Universal Robots PolyScope program: Subprogram .urp

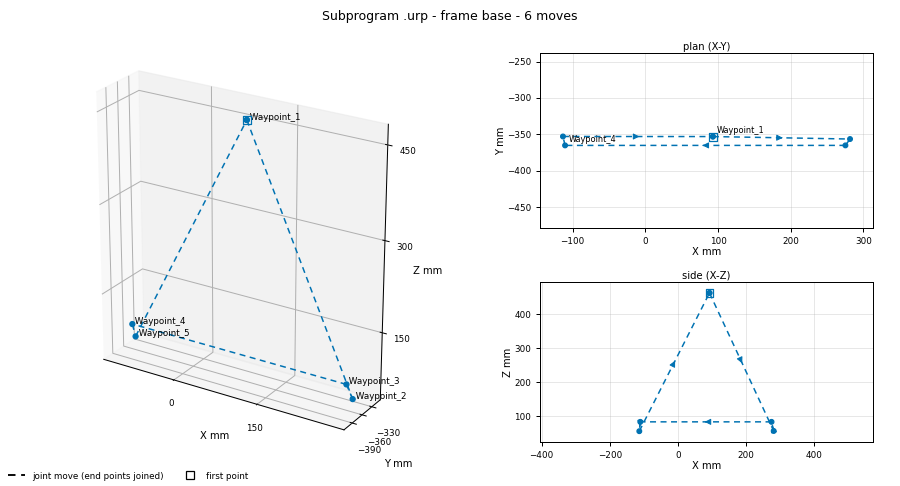
[picture p0: tool path of Subprogram .urp in frame base, 6 of 6 moves have a stored position in this frame; points joined in program order, loops and branches not executed]
Program PythonSubprogram  (installation=default directory=/programs/usbdisk/NoodleBotSoftware createdIn=3.12.1.90940 lastSavedIn=3.12.1.90940 robotSerialNumber=2017354841)
Calibrated DH parameters: a=[0.000094, -0.006117, -0.382762, 0.000086, 0.000044, 0]; d=[0.089236, 217.751846, -204.357806, -13.283746, 0.094902, 0.082641]; alpha=[1.57017, 0.001953, -0.006493, 1.570192, -1.570543, 0]; deltaTheta=[0.000036, 1.556386, -1.779789, 0.223359, -0.000014, -0.000001]
BeforeStart
  var_1 := socket_open("192.168.0.100",30000)
Robot Program (runOnlyOnce=false)
  Loop While (checkContinuously=false) expression=var_1≟ False
    var_1 := socket_open("192.168.0.100",30000)
    Wait Sleep waitTime=0.5
  Script: socket_send_string("asking_for_data")
  Wait Sleep waitTime=0.5
  var_2 := socket_read_ascii_float(1)
  Wait Sleep waitTime=0.5
  var_1 := False
  Script: socket_close()
  If var_2[0]≟1
    Call Test_ur5a
SubProgram -> Test_ur5a
SubProgram Test_ur5a (keepSynchronizedWithDisk=false) programFile=/programs/Test ur5a.urp
  MoveJ speed 60 deg/s, acceleration 80 deg/s^2 (useActiveTCP=true)
    URCap RG2 (RG - On Robot, OnRobot A/S) dataModel(depthCompensate=false, force=40, payload=0.0, width=86, name=RG2(86))
    Waypoint Waypoint_1: TCP in base x=92.939 y=-353.097 z=462.595 mm, rx=1.1692 ry=-1.2408 rz=1.1709 rad; joints [88.542, -137.018, 138.65, 178.588, 268.341, 89.999] deg; flange x=103.097 y=-166.778 z=463.297 mm, rx=1.2543 ry=1.1818 rz=-1.2438 rad
    Wait Sleep waitTime=1
    Waypoint Waypoint_2: TCP in base x=281.568 y=-356.493 z=57.062 mm, rx=2.4509 ry=-1.0812 rz=-0.3973 rad; joints [131.142, -83.255, 116.241, 241.937, 240.139, 90.003] deg; flange x=360.116 y=-306.414 z=218.729 mm, rx=-1.1245 ry=-2.5488 rz=0.6202 rad
    URCap RG2 (RG - On Robot, OnRobot A/S) dataModel(depthCompensate=false, payload=0.0, force=40, width=0, name=RG2(0))
    Wait Sleep waitTime=1
    Waypoint Waypoint_3: motionParameters(jointSpeed=1.745329 jointAcceleration=4.363323 cartesianSpeed=0.25 cartesianAcceleration=1.2); TCP in base x=275.23 y=-365.244 z=83.858 mm, rx=2.4082 ry=-1.0628 rz=-0.4074 rad; joints [131.131, -84.8, 114.576, 244.685, 237.533, 90.016] deg; flange x=358.189 y=-309.185 z=241.34 mm, rx=-1.1149 ry=-2.5256 rz=0.6807 rad
    Wait Sleep waitTime=1
    Waypoint Waypoint_4: motionParameters(jointSpeed=1.745329 jointAcceleration=4.363323 cartesianSpeed=0.25 cartesianAcceleration=1.2); TCP in base x=-110.35 y=-365.263 z=83.889 mm, rx=2.4083 ry=-1.0627 rz=-0.4074 rad; joints [69.173, -109.993, 144.496, 207.947, 251.859, 22.112] deg; flange x=-27.414 y=-309.154 z=241.302 mm, rx=-1.1146 ry=-2.5256 rz=0.6805 rad
    Waypoint Waypoint_5: TCP in base x=-113.251 y=-352.97 z=56.401 mm, rx=2.4743 ry=-1.0833 rz=-0.4569 rad; joints [69.146, -107.002, 145.454, 208.35, 250.31, 22.145] deg; flange x=-30.387 y=-310.642 z=218.159 mm, rx=-1.1049 ry=-2.5237 rz=0.5697 rad
    URCap RG2 (RG - On Robot, OnRobot A/S) dataModel(depthCompensate=false, force=40, payload=0.0, width=70, name=RG2(70))
    Waypoint Waypoint_1: TCP in base x=92.939 y=-353.097 z=462.595 mm, rx=1.1692 ry=-1.2408 rz=1.1709 rad; joints [88.542, -137.018, 138.65, 178.588, 268.341, 89.999] deg; flange x=103.097 y=-166.778 z=463.297 mm, rx=1.2543 ry=1.1818 rz=-1.2438 rad
